VAR_GLOBAL
  MixerRenamed : FB_Device;
  FlowValue : REAL;
  NewlyAddedSensor : INT;
  ValveCommand : BOOL := FALSE;
END_VAR
